PROGRAM MAIN_CONVAYOR
VAR
	inc: INT:=1;
	temp: INT;
	state: INT:=0;
	total_length: INT;
	cart_space: INT;
	cornerX: INT;
	cornerY: INT;
	bMOVE:BOOL :=FALSE;
	bSTARTUP: BOOL:=FALSE;
	rtrigNext: R_TRIG;
	counter: INT;
	tNext: TON;
	tDelay: TON;
	bDELAY: BOOL:=FALSE;
	first_run: BOOL:=FALSE;
END_VAR

FOR counter:=1 TO num_of_carts BY 1 DO
	fbCART[counter]();
END_FOR;

IF NOT first_run THEN
	A_set_cart_spaces();
	A_SETUP();
	first_run:=TRUE;
END_IF



tDelay(IN:=bDELAY);
tNext(IN:=bMOVE , PT:=T#1S , Q=> , ET=> );

CASE eMAIN_CONVAYOR_STATE OF
	E_CONVAYOR_STATE.uninit:
		A_SETUP();
		eMAIN_CONVAYOR_STATE:=E_CONVAYOR_STATE.idle;
	
	E_CONVAYOR_STATE.idle:
		bDELAY:=FALSE;
		bMOVE:=FALSE;
		bCONV_MAIN_INPOS:=TRUE;
	
	E_CONVAYOR_STATE.do_move: // open advance piston and update carts
		IF bCONV_MAIN_INPOS THEN		 
			A_CARTS_STEP();
			fbPISTON[13].A_OPEN();
			bCONV_MAIN_INPOS:=FALSE;
		END_IF
		bMOVE:=TRUE;
		bCONV_MAIN_INPOS:=FALSE;
		IF fbPISTON[13].PistonStatus= ePistonStatus.OPENED THEN
			A_CARTS_STEP();
			bMOVE:=FALSE;
			bCONV_MAIN_INPOS:=TRUE;
			eMAIN_CONVAYOR_STATE:=E_CONVAYOR_STATE.st1;
		END_IF
	
	E_CONVAYOR_STATE.st1://delay and close advansed piston
		tDELAY.PT:=T#0.6S;
		bDELAY:=TRUE;
		IF tDelay.Q THEN
			fbPISTON[13].A_CLOSE();
			eMAIN_CONVAYOR_STATE:=E_CONVAYOR_STATE.done;
		END_IF
		IF fbPISTON[13].PistonStatus= ePistonStatus.CLOSED THEN
			//...
		END_IF		
	
	E_CONVAYOR_STATE.done:
		//...
	
	E_CONVAYOR_STATE.pause:
	//paused
	
END_CASE

ACTION A_CARTS_STEP:
FOR counter:=1 TO num_of_carts BY 1 DO
	fbCART[counter].A_STEP();
END_FOR;
END_ACTION

ACTION A_set_cart_spaces:
 total_length := (conv_height*2)+(conv_length*2);
cart_space := total_length /((num_of_carts*2));
inc:=1;
posArrX[inc]:= 0+X_OFFSET;
posArrY[inc]:= 0+(conv_height/2)+Y_OFFSET;



WHILE state = 0 DO    //left1
	IF posArrY[inc]-cart_space < Y_OFFSET THEN
		temp :=cart_space - (posArrY[inc]-Y_OFFSET);
		posArrX[inc+1]:= temp+X_OFFSET;
		posArrY[inc+1]:= 0+Y_OFFSET;
		state:=1;
	ELSE
		posArrX[inc+1]:= 0+X_OFFSET;
		posArrY[inc+1]:=posArrY[inc]- cart_space;
		inc :=inc+1;
	END_IF
END_WHILE
inc := inc+1;

WHILE state = 1 DO // top
	IF posArrX[inc]+cart_space > (X_OFFSET+conv_length) THEN
		temp :=cart_space - ((X_OFFSET+conv_length)-posArrX[inc]);
		posArrX[inc+1]:= conv_length+X_OFFSET;
		posArrY[inc+1]:= temp+Y_OFFSET;
		state:=2;
	ELSE
		posArrX[inc+1]:= posArrX[inc]+cart_space;
		posArrY[inc+1]:=Y_OFFSET;
		inc :=inc+1;
	END_IF
END_WHILE
inc :=inc+1;	

WHILE state = 2 DO // right
	IF posArrY[inc]+cart_space > (Y_OFFSET+conv_height) THEN
		temp :=cart_space - ((Y_OFFSET+conv_height)-posArrY[inc]);
		posArrX[inc+1]:= (conv_length+X_OFFSET)-temp;
		posArrY[inc+1]:= 0+Y_OFFSET+conv_height;
		state:=3;
	ELSE
		posArrX[inc+1]:= 0+X_OFFSET+conv_length;
		posArrY[inc+1]:=posArrY[inc]+ cart_space;
		inc :=inc+1;
	END_IF	
END_WHILE
inc :=inc+1;	

WHILE state = 3 DO //bottom
	IF  posArrX[inc]-cart_space < X_OFFSET THEN
		temp :=cart_space - (posArrX[inc]-X_OFFSET);
		posArrX[inc+1]:= X_OFFSET;
		posArrY[inc+1]:= Y_OFFSET+ conv_height-temp;
		state:=4;
	ELSE
		posArrX[inc+1]:= posArrX[inc]-cart_space;
		posArrY[inc+1]:=Y_OFFSET+conv_height;
		inc :=inc+1;
		
	END_IF
END_WHILE

IF inc > 34 THEN
	RETURN;
END_IF


inc :=inc+1;

WHILE state = 4 DO    //left2
	IF posArrY[inc]-cart_space < ((conv_height/2)+Y_OFFSET) THEN
		state:=5;
	ELSE
		posArrX[inc+1]:= 0+X_OFFSET;
		posArrY[inc+1]:=posArrY[inc]- cart_space;
		inc :=inc+1;
		
	END_IF
END_WHILE
END_ACTION

ACTION A_SETUP:
	bSTARTUP:=TRUE;
	fbCART[1].stCART.position:=1;
	fbCART[1].stCART.color:=1;
	fbCART[1].stCART.nNAME:=INT_TO_STRING(1001);
	fbCART[1].stCART.posX:=posArrX[1];
	fbCART[1].stCART.posY:=posArrY[1];
		
	FOR counter:=1 TO (num_of_carts-1) BY 1 DO
		fbCART[counter+1].stCART.position:=37-((counter*2));
		fbCART[counter+1].stCART.color:=1;
		fbCART[counter+1].stCART.nNAME:=INT_TO_STRING(1000+counter+1);
		fbCART[counter+1].stCART.posX:=posArrX[37-((counter*2))];
		fbCART[counter+1].stCART.posY:=posArrY[37-((counter*2))];
	END_FOR;
END_ACTION

END_PROGRAM

(* stored: Version 1.1.0.1, ProductVersion 3.1.4024.12
   POU MAIN_CONVAYOR: Id {230d7160-cfd8-4561-bda5-963e513f3cc2}, SpecialFunc None
   Action A_CARTS_STEP: Id {7a1e55b7-d701-499d-a448-d86c230d8eaf}
   Action A_set_cart_spaces: Id {7d4d76aa-d053-4a28-a62b-1eb33cb8ead7}
   Action A_SETUP: Id {743a8297-84d8-4da3-9839-4637b3eb1bf1} *)
